Staubli VAL3: cycle_pause.pgx

program cycle_pause()
begin
  //
  // PAUSE THE CYCLE
  //
  if !cycleStatus:bPause
    logMsg("[KERNEL] PLC:pause cycle")
    // pause
    cycleStatus:bToPause=true
    watch(cycleStatus:bToPause==false,1)
    //
  endIf
  //
end
